// TIA Portal V20 export
TYPE "LER_TypeFATMode_HoursTest_ProcessValue"
// stored: Access Published
   STRUCT
      ProcTimeLeft : Time;
      SelectHours_ProcessValue : Time;
   END_STRUCT;
END_TYPE
